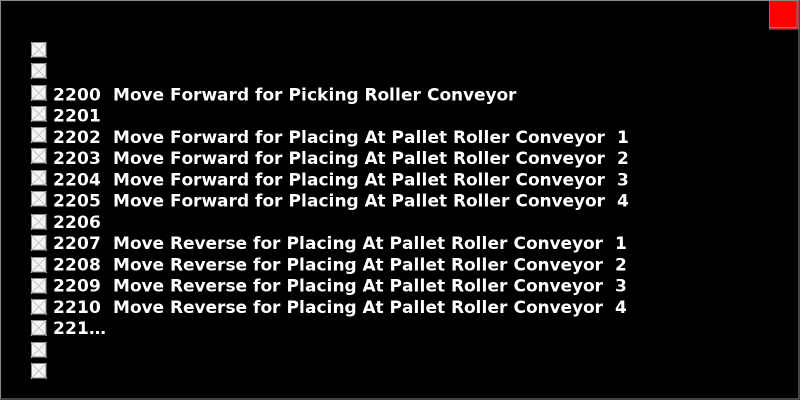
VISUALIZATION P1_DO2  // 800x400, background image 
    ImageSwitcher (31,42 15x15), variable: InputOutput_GVL.xIn1000, behaviour: TOGGLE
    Label (50,16 625x391), "2200 Move Forward for Picking Roller Conveyor 2201 2202 Move Forward for Placing At Pallet Roller Conveyor 1 2203 Move Forward for Placing At Pallet Roller Conveyor 2 2204 Move Forward for Placing At Pallet Roller Conveyor 3 2205 Move Forward for Placing At Pallet Roller Conveyor 4 2206 2207 Move Reverse for Placing At Pallet Roller Conveyor 1 2208 Move Reverse for Placing At Pallet Roller Conveyor 2 2209 Move Reverse for Placing At Pallet Roller Conveyor 3 2210 Move Reverse for Placing At Pallet Roller Conveyor 4 2211 2212 2213 2214 2215 Reset Error for All Inverter at P1, Relay"
    ImageSwitcher (31,63 15x15), variable: InputOutput_GVL.xIn1001, behaviour: TOGGLE
    ImageSwitcher (31,85 15x15), variable: InputOutput_GVL.xIn1002, behaviour: TOGGLE
    ImageSwitcher (31,106 15x15), variable: InputOutput_GVL.xIn1003, behaviour: TOGGLE
    ImageSwitcher (31,127 15x15), variable: InputOutput_GVL.xIn1004, behaviour: TOGGLE
    ImageSwitcher (31,148 15x15), variable: InputOutput_GVL.xIn1005, behaviour: TOGGLE
    ImageSwitcher (31,170 15x15), variable: InputOutput_GVL.xIn1006, behaviour: TOGGLE
    ImageSwitcher (31,191 15x15), variable: InputOutput_GVL.xIn1007, behaviour: TOGGLE
    ImageSwitcher (31,214 15x15), variable: InputOutput_GVL.xIn1008, behaviour: TOGGLE
    ImageSwitcher (31,235 15x15), variable: InputOutput_GVL.xIn1009, behaviour: TOGGLE
    ImageSwitcher (31,257 15x15), variable: InputOutput_GVL.xIn1010, behaviour: TOGGLE
    ImageSwitcher (31,278 15x15), variable: InputOutput_GVL.xIn1011, behaviour: TOGGLE
    ImageSwitcher (31,299 15x15), variable: InputOutput_GVL.xIn1012, behaviour: TOGGLE
    ImageSwitcher (31,320 15x15), variable: InputOutput_GVL.xIn1013, behaviour: TOGGLE
    ImageSwitcher (31,342 15x15), variable: InputOutput_GVL.xIn1014, behaviour: TOGGLE
    ImageSwitcher (31,363 15x15), variable: InputOutput_GVL.xIn1015, behaviour: TOGGLE
    Button (769,-1 30x30), image: VisuSymbols.Symbols.Wrong
        OnMouseClick: CloseDialog Dialog=P1_DO2, Result=OK, NumpadKeypadSet=True
END_VISUALIZATION

(* stored: Version 1.1.0.1, ProductVersion 3.1.4024.12
   Visu P1_DO2: Id {dc34234f-9daa-4b4c-baae-4796567c6a3e} *)
